FUNCTION_BLOCK TEST_LTN (* Test LT functions of numerical values *)
  (* Standard: IEC 61499-1 *)
  (* Version 0.0, 2006-09-11, JHC, Holobloc Inc *)
  (* Compiler header: package fb.rt.test; *)
  (* Compiler classdef: SimpleFB *)
  (* Compiler Java Sun JDK 1.5.0 *)
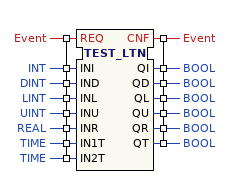
  EVENT_INPUT
    REQ WITH INI, INL, INU, IND, INR, IN1T, IN2T;
  END_EVENT
  EVENT_OUTPUT
    CNF WITH QI, QD, QL, QU, QR, QT;
  END_EVENT
  VAR_INPUT
    INI : INT;
    IND : DINT;
    INL : LINT;
    INU : UINT;
    INR : REAL;
    IN1T : TIME;
    IN2T : TIME;
  END_VAR
  VAR_OUTPUT
    QI : BOOL;
    QD : BOOL;
    QL : BOOL;
    QU : BOOL;
    QR : BOOL;
    QT : BOOL;
  END_VAR
  ALGORITHM REQ IN FBD:
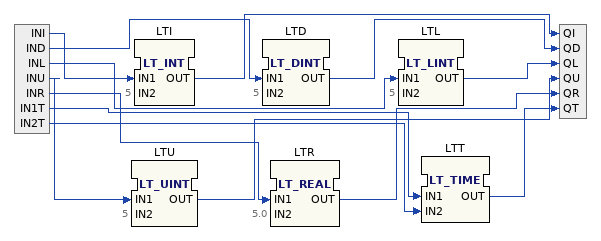
    FBS
      LTI : LT_INT(IN2 := 5);
      LTD : LT_DINT(IN2 := 5);
      LTL : LT_LINT(IN2 := 5);
      LTU : LT_UINT(IN2 := 5);
      LTR : LT_REAL(IN2 := 5.0);
      LTT : LT_TIME;
    END_FBS
    DATA_CONNECTIONS
      INI TO LTI.IN1;
      IND TO LTD.IN1;
      INL TO LTL.IN1;
      INU TO LTU.IN1;
      INR TO LTR.IN1;
      LTI.OUT TO QI;
      LTD.OUT TO QD;
      LTL.OUT TO QL;
      LTU.OUT TO QU;
      LTR.OUT TO QR;
      LTT.OUT TO QT;
      IN1T TO LTT.IN1;
      IN2T TO LTT.IN2;
    END_CONNECTIONS
  END_ALGORITHM
END_FUNCTION_BLOCK
